Staubli VAL3: taskKiller.pgx

program taskKiller(string sTask_)
begin
    //
  //\param sTask_
  //
taskKill(sTask_)
end
